(* PLC project Sin nombre, Desconocido Sin nombre 1 *)
(* stored: creationDateTime 2022-10-17T16:56:25, modificationDateTime 2022-10-17T18:05:40 *)

PROGRAM program0
  VAR
    Out1 AT %QX0.0 : BOOL := 0;
  END_VAR
  VAR
    TRU : BOOL := 1;
    TP0 : TP;
  END_VAR

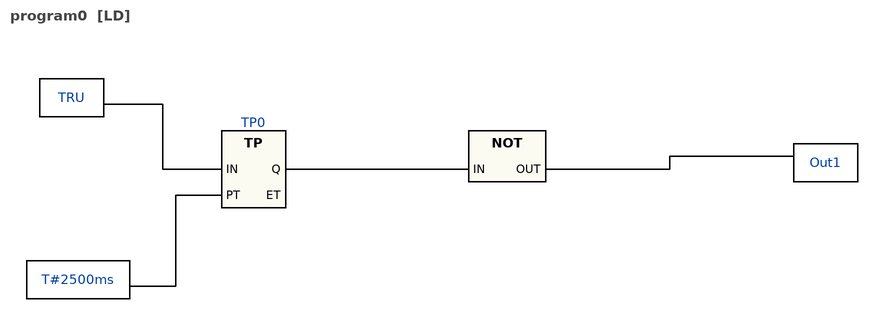
(* LD diagram, written out as Structured Text *)
TP0(IN := TRU, PT := T#2500ms);
Out1 := NOT TP0.Q;
END_PROGRAM

CONFIGURATION Config0
  RESOURCE Res0 ON PLC
    TASK task0(INTERVAL := T#20ms, PRIORITY := 0);
    PROGRAM instance0 WITH task0 : program0;
  END_RESOURCE
END_CONFIGURATION
